(* IEC 61131-3 sources: SIGMATEK-Jumag-Utils-Examples/typeManipulation/Class/mergeBSINT, 1 file *)

(* ---- mergeBSINT.st ---- *)
(*!
<Class
	Name               = "mergeBSINT"
	Revision           = "0.0"
	RealtimeTask       = "false"
	CyclicTask         = "true"
	DefCyclictime      = "10 ms"
	BackgroundTask     = "false"
	Sigmatek           = "false"
	OSInterface        = "false"
	HighPriority       = "false"
	Automatic          = "false"
	UpdateMode         = "Prescan"
	SharedCommandTable = "true"
	Objectsize         = "(284,120)">
	<Channels>
		<Server Name="ClassSvr" Visualized="false" Initialize="false" WriteProtected="true" Retentive="false"/>
		<Server Name="LSB" Visualized="false" Initialize="true" WriteProtected="false" Retentive="false"/>
		<Server Name="merged" Visualized="false" Initialize="false" WriteProtected="true" Retentive="false"/>
		<Server Name="MSB" Visualized="false" Initialize="true" WriteProtected="false" Retentive="false"/>
	</Channels>
	<Dependencies>
		<Files>
			<File Path=".\Source\typeManipulation.c"/>
		</Files>
	</Dependencies>
</Class>
*)
mergeBSINT : CLASS
  //Servers:
	ClassSvr 	: SvrChCmd_DINT;
	merged 	: SvrCh_DINT;
	MSB 	: SvrCh_DINT;
	LSB 	: SvrCh_DINT;
  //Clients:
  //Variables:
  //Functions:

	FUNCTION VIRTUAL GLOBAL CyWork
		VAR_INPUT
			EAX 	: UDINT;
		END_VAR
		VAR_OUTPUT
			state (EAX) 	: UDINT;
		END_VAR;
  //Tables:
	FUNCTION @STD
		VAR_OUTPUT
			ret_code	: CONFSTATES;
		END_VAR;
	FUNCTION GLOBAL TAB @CT_;
END_CLASS;

Function Global __cdecl mergeBSINT
VAR_INPUT
  MSB : BSINT;
  LSB : BSINT;
END_VAR
VAR_OUTPUT
  Q : UINT;
END_VAR;

FUNCTION VIRTUAL GLOBAL mergeBSINT::CyWork
	VAR_INPUT
		EAX 	: UDINT;
	END_VAR
	VAR_OUTPUT
		state (EAX) 	: UDINT;
	END_VAR

  merged := mergeBSINT(MSB:=to_usint(MSB), LSB:=to_usint(LSB));

	state := READY;

END_FUNCTION
